(* CODESYS project CODESYS_GIT
   Project Profile: MachineProfile

Project tree, tasks and I/O mapping:
  Device : XP340, Beijer Electronics, order no. XP340, version 1.3.40.200
    application Application
      libraries: NextoStandard, 1.3.0.1 (WAA); LibDataTypes, 1.0.0.0 (Manufacturer); LibIntegratedIo, 1.0.0.16 (Manufacturer); CmpApp, 3.5.17.0 (System); 3SLicense, 3.5.17.0 (3S - Smart Software Solutions GmbH); XP340 Diagnostic Structs, 1.0.0.4 (Manufacturer)
      task MainTask (cyclic, interval 20 ms, priority 13, watchdog 1000 ms x 1) calls MainPrg
      SystemEvents/
        function Prepare_Start [ST]
        function Prepare_Stop [ST]
        function Start_Done [ST]
        function Stop_Done [ST]
      SystemGVLs/
        global variables IntegratedIO
        global variables Special_Variables
        global variables System_Diagnostics
      SystemPOUs/
        program MainPrg [ST]
        program SpecialVariablesPrg [ST]
      UserGVLs/
        global variables Disables
        global variables Qualities
        global variables ReqDiagnostics
      UserPOUs/
        program StartPrg [ST]
        program UserPrg [ST]
    Configuration : Config, WAA, order no. Configuration, version 1.1.1.3
        settings: Machine Profile = TRUE
      XP340 : XP340, Beijer Electronics, order no. XP340, version 1.3.40.200
          settings: DC sync0 cycletime = 5000; IOModule's Address for interrupt = 255; CurrentProjectProfileParameter = 'MachineProfile'
        <Empty>
        CAN
        COM 1
        Integrated I/O
            settings: Parameter list definition.Count = 16; Item_00000.Index = 0; Item_00000.Variable = 'I00'; Item_00000.Data Type = 'BOOL'; Item_00000.Channel = 'Input 00 '; Item_00000.Description = 'Digital Input 00 '; Item_00001.Index = 1; Item_00001.Variable = 'I01'; Item_00001.Data Type = 'BOOL'; Item_00001.Channel = 'Input 01 '; Item_00001.Description = 'Digital Input 01 '; Item_00002.Index = 2; Item_00002.Variable = 'I02'; Item_00002.Data Type = 'BOOL'; Item_00002.Channel = 'Input 02 '; Item_00002.Description = 'Digital Input 02 '; Item_00003.Index = 3; Item_00003.Variable = 'I03'; Item_00003.Data Type = 'BOOL'; Item_00003.Channel = 'Input 03 '; Item_00003.Description = 'Digital Input 03 '; Item_00004.Index = 4; Item_00004.Variable = 'I04'; Item_00004.Data Type = 'BOOL'; Item_00004.Channel = 'Input 04 '; Item_00004.Description = 'Digital Input 04 '; Item_00005.Index = 5; Item_00005.Variable = 'I05'; Item_00005.Data Type = 'BOOL'; Item_00005.Channel = 'Input 05 '; Item_00005.Description = 'Digital Input 05 '; Item_00006.Index = 6; Item_00006.Variable = 'I06'; Item_00006.Data Type = 'BOOL'; Item_00006.Channel = 'Input 06 '; Item_00006.Description = 'Digital Input 06 '; Item_00007.Index = 7; Item_00007.Variable = 'I07'; Item_00007.Data Type = 'BOOL'; Item_00007.Channel = 'Input 07 ';
              Item_00007.Description = 'Digital Input 07 '; Item_00008.Index = 8; Item_00008.Variable = 'I10'; Item_00008.Data Type = 'BOOL'; Item_00008.Channel = 'Input 10 '; Item_00008.Description = 'Digital Input 10 '; Item_00009.Index = 9; Item_00009.Variable = 'I11'; Item_00009.Data Type = 'BOOL'; Item_00009.Channel = 'Input 11 '; Item_00009.Description = 'Digital Input 11 '; Item_00010.Index = 10; Item_00010.Variable = 'I12'; Item_00010.Data Type = 'BOOL'; Item_00010.Channel = 'Input 12 '; Item_00010.Description = 'Digital Input 12 '; Item_00011.Index = 11; Item_00011.Variable = 'I13'; Item_00011.Data Type = 'BOOL'; Item_00011.Channel = 'Input 13 '; Item_00011.Description = 'Digital Input 13 '; Item_00012.Index = 12; Item_00012.Variable = 'I14'; Item_00012.Data Type = 'BOOL'; Item_00012.Channel = 'Input 14 '; Item_00012.Description = 'Digital Input 14 '; Item_00013.Index = 13; Item_00013.Variable = 'I15'; Item_00013.Data Type = 'BOOL'; Item_00013.Channel = 'Input 15 '; Item_00013.Description = 'Digital Input 15 '; Item_00014.Index = 14; Item_00014.Variable = 'I16'; Item_00014.Data Type = 'BOOL'; Item_00014.Channel = 'Input 16 '; Item_00014.Description = 'Digital Input 16 '; Item_00015.Index = 15; Item_00015.Variable = 'I17'; Item_00015.Data Type = 'BOOL'; Item_00015.Channel = 'Input 17 ';
              Item_00015.Description = 'Digital Input 17 '; Parameter list definition.Count = 16; Item_00000.Index = 0; Item_00000.Variable = 'Q00'; Item_00000.Data Type = 'BOOL'; Item_00000.Channel = 'Output 00 '; Item_00000.Description = 'Digital Output 00 '; Item_00001.Index = 1; Item_00001.Variable = 'Q01'; Item_00001.Data Type = 'BOOL'; Item_00001.Channel = 'Output 01 '; Item_00001.Description = 'Digital Output 01 '; Item_00002.Index = 2; Item_00002.Variable = 'Q02'; Item_00002.Data Type = 'BOOL'; Item_00002.Channel = 'Output 02 '; Item_00002.Description = 'Digital Output 02 '; Item_00003.Index = 3; Item_00003.Variable = 'Q03'; Item_00003.Data Type = 'BOOL'; Item_00003.Channel = 'Output 03 '; Item_00003.Description = 'Digital Output 03 '; Item_00004.Index = 4; Item_00004.Variable = 'Q04'; Item_00004.Data Type = 'BOOL'; Item_00004.Channel = 'Output 04 '; Item_00004.Description = 'Digital Output 04 '; Item_00005.Index = 5; Item_00005.Variable = 'Q05'; Item_00005.Data Type = 'BOOL'; Item_00005.Channel = 'Output 05 '; Item_00005.Description = 'Digital Output 05 '; Item_00006.Index = 6; Item_00006.Variable = 'Q06'; Item_00006.Data Type = 'BOOL'; Item_00006.Channel = 'Output 06 '; Item_00006.Description = 'Digital Output 06 '; Item_00007.Index = 7; Item_00007.Variable = 'Q07'; Item_00007.Data Type = 'BOOL';
              Item_00007.Channel = 'Output 07 '; Item_00007.Description = 'Digital Output 07 '; Item_00008.Index = 8; Item_00008.Variable = 'Q10'; Item_00008.Data Type = 'BOOL'; Item_00008.Channel = 'Output 10 '; Item_00008.Description = 'Digital Output 10 '; Item_00009.Index = 9; Item_00009.Variable = 'Q11'; Item_00009.Data Type = 'BOOL'; Item_00009.Channel = 'Output 11 '; Item_00009.Description = 'Digital Output 11 '; Item_00010.Index = 10; Item_00010.Variable = 'Q12'; Item_00010.Data Type = 'BOOL'; Item_00010.Channel = 'Output 12 '; Item_00010.Description = 'Digital Output 12 '; Item_00011.Index = 11; Item_00011.Variable = 'Q13'; Item_00011.Data Type = 'BOOL'; Item_00011.Channel = 'Output 13 '; Item_00011.Description = 'Digital Output 13 '; Item_00012.Index = 12; Item_00012.Variable = 'Q14'; Item_00012.Data Type = 'BOOL'; Item_00012.Channel = 'Output 14 '; Item_00012.Description = 'Digital Output 14 '; Item_00013.Index = 13; Item_00013.Variable = 'Q15'; Item_00013.Data Type = 'BOOL'; Item_00013.Channel = 'Output 15 '; Item_00013.Description = 'Digital Output 15 '; Item_00014.Index = 14; Item_00014.Variable = 'Q16'; Item_00014.Data Type = 'BOOL'; Item_00014.Channel = 'Output 16 '; Item_00014.Description = 'Digital Output 16 '; Item_00015.Index = 15; Item_00015.Variable = 'Q17'; Item_00015.Data Type = 'BOOL';
              Item_00015.Channel = 'Output 17 '; Item_00015.Description = 'Digital Output 17 '; Parameter list definition.Count = 5; Item_00000.Index = 0; Item_00000.Variable = 'AI0'; Item_00000.Data Type = 'INT'; Item_00000.Channel = 'Analog Input 0 '; Item_00000.Description = 'Analog Input 0 '; Item_00001.Index = 1; Item_00001.Variable = 'AI1'; Item_00001.Data Type = 'INT'; Item_00001.Channel = 'Analog Input 1 '; Item_00001.Description = 'Analog Input 1 '; Item_00002.Index = 2; Item_00002.Variable = 'AI2'; Item_00002.Data Type = 'INT'; Item_00002.Channel = 'Analog Input 2 '; Item_00002.Description = 'Analog Input 2 '; Item_00003.Index = 3; Item_00003.Variable = 'AI3'; Item_00003.Data Type = 'INT'; Item_00003.Channel = 'Analog Input 3 '; Item_00003.Description = 'Analog Input 3 '; Item_00004.Index = 4; Item_00004.Variable = 'AI4'; Item_00004.Data Type = 'INT'; Item_00004.Channel = 'Analog Input 4 '; Item_00004.Description = 'Analog Input 4 '; Parameter list definition.Count = 4; Item_00000.Index = 0; Item_00000.Variable = 'AO0'; Item_00000.Data Type = 'INT'; Item_00000.Channel = 'Analog Output 0 '; Item_00000.Description = 'Analog Output 0 '; Item_00001.Index = 1; Item_00001.Variable = 'AO1'; Item_00001.Data Type = 'INT'; Item_00001.Channel = 'Analog Output 1 '; Item_00001.Description = 'Analog Output 1 '; Item_00002.Index = 2;
              Item_00002.Variable = 'AO2'; Item_00002.Data Type = 'INT'; Item_00002.Channel = 'Analog Output 2 '; Item_00002.Description = 'Analog Output 2 '; Item_00003.Index = 3; Item_00003.Variable = 'AO3'; Item_00003.Data Type = 'INT'; Item_00003.Channel = 'Analog Output 3 '; Item_00003.Description = 'Analog Output 3 '; Parameter list definition.Count = 2; Item_00000.Index = 0; Item_00000.Variable = 'RI0'; Item_00000.Data Type = 'INT'; Item_00000.Channel = 'RTD Input 0 '; Item_00000.Description = 'RTD Input 0 '; Item_00001.Index = 1; Item_00001.Variable = 'RI1'; Item_00001.Data Type = 'INT'; Item_00001.Channel = 'RTD Input 1 '; Item_00001.Description = 'RTD Input 1 '
        NET 1
*)

// Device/Application/SystemGVLs/IntegratedIO
VAR_GLOBAL

	// Structured tags for I/O points
	DigitalInputs  : T_DIGITAL_INPUTS_1;                        // Digital Inputs structure
	DigitalOutputs : T_DIGITAL_OUTPUTS_1;                       // Digital Outputs structure
	FastInputs     : T_FAST_INPUTS_1;                           // Fast Inputs structure
	FastOutputs    : T_FAST_OUTPUTS_1;                          // Fast Outputs structure
	AnalogInputs   : T_ANALOG_INPUTS_1;                         // Analog Inputs structure
	AnalogOutputs  : T_ANALOG_OUTPUTS_1;                        // Analog Ouputs structure
	RtdInputs      : T_RTD_INPUTS_1;                            // RTD Inputs structure

	// Direct tags for I/O points
	I00            : REFERENCE TO BOOL   := DigitalInputs.I00;  // Digital Input 00 
	I01            : REFERENCE TO BOOL   := DigitalInputs.I01;  // Digital Input 01 
	I02            : REFERENCE TO BOOL   := DigitalInputs.I02;  // Digital Input 02 
	I03            : REFERENCE TO BOOL   := DigitalInputs.I03;  // Digital Input 03 
	I04            : REFERENCE TO BOOL   := DigitalInputs.I04;  // Digital Input 04 
	I05            : REFERENCE TO BOOL   := DigitalInputs.I05;  // Digital Input 05 
	I06            : REFERENCE TO BOOL   := DigitalInputs.I06;  // Digital Input 06 
	I07            : REFERENCE TO BOOL   := DigitalInputs.I07;  // Digital Input 07 
	I10            : REFERENCE TO BOOL   := DigitalInputs.I10;  // Digital Input 10 
	I11            : REFERENCE TO BOOL   := DigitalInputs.I11;  // Digital Input 11 
	I12            : REFERENCE TO BOOL   := DigitalInputs.I12;  // Digital Input 12 
	I13            : REFERENCE TO BOOL   := DigitalInputs.I13;  // Digital Input 13 
	I14            : REFERENCE TO BOOL   := DigitalInputs.I14;  // Digital Input 14 
	I15            : REFERENCE TO BOOL   := DigitalInputs.I15;  // Digital Input 15 
	I16            : REFERENCE TO BOOL   := DigitalInputs.I16;  // Digital Input 16 
	I17            : REFERENCE TO BOOL   := DigitalInputs.I17;  // Digital Input 17 

	Q00            : REFERENCE TO BOOL   := DigitalOutputs.Q00; // Digital Output 00 
	Q01            : REFERENCE TO BOOL   := DigitalOutputs.Q01; // Digital Output 01 
	Q02            : REFERENCE TO BOOL   := DigitalOutputs.Q02; // Digital Output 02 
	Q03            : REFERENCE TO BOOL   := DigitalOutputs.Q03; // Digital Output 03 
	Q04            : REFERENCE TO BOOL   := DigitalOutputs.Q04; // Digital Output 04 
	Q05            : REFERENCE TO BOOL   := DigitalOutputs.Q05; // Digital Output 05 
	Q06            : REFERENCE TO BOOL   := DigitalOutputs.Q06; // Digital Output 06 
	Q07            : REFERENCE TO BOOL   := DigitalOutputs.Q07; // Digital Output 07 
	Q10            : REFERENCE TO BOOL   := DigitalOutputs.Q10; // Digital Output 10 
	Q11            : REFERENCE TO BOOL   := DigitalOutputs.Q11; // Digital Output 11 
	Q12            : REFERENCE TO BOOL   := DigitalOutputs.Q12; // Digital Output 12 
	Q13            : REFERENCE TO BOOL   := DigitalOutputs.Q13; // Digital Output 13 
	Q14            : REFERENCE TO BOOL   := DigitalOutputs.Q14; // Digital Output 14 
	Q15            : REFERENCE TO BOOL   := DigitalOutputs.Q15; // Digital Output 15 
	Q16            : REFERENCE TO BOOL   := DigitalOutputs.Q16; // Digital Output 16 
	Q17            : REFERENCE TO BOOL   := DigitalOutputs.Q17; // Digital Output 17 

	AI0            : REFERENCE TO INT    := AnalogInputs.AI0;   // Analog Input 0 
	AI1            : REFERENCE TO INT    := AnalogInputs.AI1;   // Analog Input 1 
	AI2            : REFERENCE TO INT    := AnalogInputs.AI2;   // Analog Input 2 
	AI3            : REFERENCE TO INT    := AnalogInputs.AI3;   // Analog Input 3 
	AI4            : REFERENCE TO INT    := AnalogInputs.AI4;   // Analog Input 4 

	AO0            : REFERENCE TO INT    := AnalogOutputs.AO0;  // Analog Output 0 
	AO1            : REFERENCE TO INT    := AnalogOutputs.AO1;  // Analog Output 1 
	AO2            : REFERENCE TO INT    := AnalogOutputs.AO2;  // Analog Output 2 
	AO3            : REFERENCE TO INT    := AnalogOutputs.AO3;  // Analog Output 3 

	RI0            : REFERENCE TO INT    := RtdInputs.RI0;      // RTD Input 0 
	RI1            : REFERENCE TO INT    := RtdInputs.RI1;      // RTD Input 1 

END_VAR

// Device/Application/SystemGVLs/Special_Variables
(*This GVL is blocked to edit.*)
VAR_GLOBAL
	Pulse_100ms : BOOL;                     //Pulse signal with 100ms period (toggles every 50ms)
	Pulse_500ms : BOOL;                     //Pulse signal with 500ms period (toggles every 250ms)
	Pulse_1s    : BOOL;                     //Pulse signal with 1s period (toggles every 500ms)
	Pulse_2s    : BOOL;                     //Pulse signal with 2s period (toggles every 1s)
	Pulse_5s    : BOOL;                     //Pulse signal with 5s period (toggles every 2,5s)
	Pulse_10s   : BOOL;                     //Pulse signal with 10s period (toggles every 5s)
	Pulse_30s   : BOOL;                     //Pulse signal with 30s period (toggles every 15s)
	Pulse_60s   : BOOL;                     //Pulse signal with 60s period (toggles every 30s)
	Pulse_Scan  : BOOL;                     //Scan pulse that toggles every MainTask cycle
	System_Time : EXTENDED_DATE_AND_TIME;   //System date and time
	Day_Of_Week : DAYS_OF_WEEK;             //Day of week
	Hour_Minute : UINT;                     //Integer variable with hour and minute (hour*100 + minute)
END_VAR

VAR_GLOBAL CONSTANT
	udiMainTaskInterval : UDINT := 20000;     //MainTask configured interval [us].
END_VAR

// Device/Application/SystemGVLs/System_Diagnostics
VAR_GLOBAL
	//DG_XP340 diagnostics variable
	DG_XP340 : T_DIAG_XP340_1;
END_VAR

// Device/Application/UserGVLs/Disables
VAR_GLOBAL
END_VAR

// Device/Application/UserGVLs/Qualities
VAR_GLOBAL
END_VAR

// Device/Application/UserGVLs/ReqDiagnostics
VAR_GLOBAL
END_VAR

// Device/Application/SystemPOUs/MainPrg
(*Main POU associated with MainTask that calls StartPrg, UserPrg/ActivePrg and NonSkippedPrg. This POU is blocked to edit.*)
PROGRAM MainPrg
VAR
   isFirstCycle : BOOL := TRUE;
END_VAR

SpecialVariablesPrg();
IF isFirstCycle THEN
   StartPrg();
   isFirstCycle := FALSE;
ELSE
   UserPrg();
END_IF;

END_PROGRAM

// Device/Application/SystemPOUs/SpecialVariablesPrg
(*This POU is blocked to edit.*)
{attribute 'hide'}
PROGRAM SpecialVariablesPrg
VAR
	udiMicroAcc:	UDINT;			// Microseconds accumulator
	uliSystemTime:	ULINT;			// System time of this cycle [us]
	uliLastSysTime:	ULINT;			// System time of last cycle [us]
END_VAR

// Save the system time of last cycle
uliLastSysTime:= uliSystemTime;

// Get system time of this cycle
SysTimeCore.SysTimeGetUs(uliSystemTime);

// Update pulse bits
IF uliLastSysTime > 0 THEN udiMicroAcc:= udiMicroAcc + ULINT_TO_UDINT(uliSystemTime - uliLastSysTime); END_IF
IF udiMicroAcc MOD 100000 >= 50000 THEN Pulse_100ms:= TRUE; ELSE Pulse_100ms:= FALSE; END_IF
IF udiMicroAcc MOD 500000 >= 250000 THEN Pulse_500ms:= TRUE; ELSE Pulse_500ms:= FALSE; END_IF
IF udiMicroAcc MOD 1000000 >= 500000 THEN Pulse_1s:= TRUE; ELSE Pulse_1s:= FALSE; END_IF
IF udiMicroAcc MOD 2000000 >= 1000000 THEN Pulse_2s:= TRUE; ELSE Pulse_2s:= FALSE; END_IF
IF udiMicroAcc MOD 5000000 >= 2500000 THEN Pulse_5s:= TRUE; ELSE Pulse_5s:= FALSE; END_IF
IF udiMicroAcc MOD 10000000 >= 5000000 THEN Pulse_10s:= TRUE; ELSE Pulse_10s:= FALSE; END_IF
IF udiMicroAcc MOD 30000000 >= 15000000 THEN Pulse_30s:= TRUE; ELSE Pulse_30s:= FALSE; END_IF
IF udiMicroAcc MOD 60000000 >= 30000000 THEN Pulse_60s:= TRUE; ELSE Pulse_60s:= FALSE; END_IF
udiMicroAcc:= udiMicroAcc MOD 120000000;

// Update scan pulse
Pulse_Scan:= NOT Pulse_Scan;

// Update system time
GetDateAndTime(System_Time);

// Update Hour_Minute
Hour_Minute:= System_Time.byHours * 100 + System_Time.byMinutes;

// Update Day of Week
Day_Of_Week:= NextoStandard.GetDayOfWeek();

END_PROGRAM

// Device/Application/UserPOUs/StartPrg
(*The code inserted by the user into this POU is executed once after startup. Before this first cycle it is not executed again. In case of redundant system, this one is executed in both CPUs during the startup.*)
PROGRAM StartPrg
VAR
END_VAR

END_PROGRAM

// Device/Application/UserPOUs/UserPrg
(*The main code inserted by the user and executed associated with the MainTask must be inserted into this POU.*)
PROGRAM UserPrg
VAR
END_VAR

END_PROGRAM

// Device/Application/SystemEvents/Prepare_Start
(*Called before application starts. Context=Communication task. Debugging=Disabled*)
FUNCTION Prepare_Start : DWORD
VAR_IN_OUT
	EventPrm: CmpApp.EVTPARAM_CmpApp;
END_VAR
VAR
END_VAR

END_FUNCTION

// Device/Application/SystemEvents/Prepare_Stop
(*Called before application stops. Context=Communication task. Debugging=Disabled*)
FUNCTION Prepare_Stop : DWORD
VAR_IN_OUT
	EventPrm: CmpApp.EVTPARAM_CmpAppStop;
END_VAR
VAR
END_VAR

END_FUNCTION

// Device/Application/SystemEvents/Start_Done
(*Called after application starts. Context=Communication task. Debugging=Disabled*)
FUNCTION Start_Done : DWORD
VAR_IN_OUT
	EventPrm: CmpApp.EVTPARAM_CmpApp;
END_VAR
VAR
END_VAR

END_FUNCTION

// Device/Application/SystemEvents/Stop_Done
(*Called after application stops. Context=Communication task. Debugging=Disabled*)
FUNCTION Stop_Done : DWORD
VAR_IN_OUT
	EventPrm: CmpApp.EVTPARAM_CmpAppStop;
END_VAR
VAR
END_VAR

END_FUNCTION
